FUNCTION_BLOCK NextFeedHorizon (* CAT Function Block Type *)
  (* Standard: 61499-2 *)
  (* Version 0.0, 7/15/2026, Schneider Electric, template *)
  PACKAGE SE.Nereda;
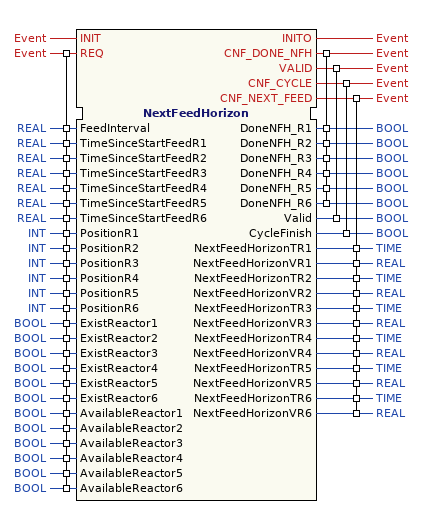
  EVENT_INPUT
    INIT;
    REQ WITH FeedInterval, TimeSinceStartFeedR1, TimeSinceStartFeedR2, TimeSinceStartFeedR3, TimeSinceStartFeedR4, TimeSinceStartFeedR5, TimeSinceStartFeedR6, PositionR1, PositionR2, PositionR3, PositionR4, PositionR5, PositionR6, ExistReactor1, ExistReactor2, ExistReactor3, ExistReactor4, ExistReactor5, ExistReactor6, AvailableReactor1, AvailableReactor2, AvailableReactor3, AvailableReactor4, AvailableReactor5, AvailableReactor6;
  END_EVENT
  EVENT_OUTPUT
    INITO;
    CNF_DONE_NFH WITH DoneNFH_R6, DoneNFH_R1, DoneNFH_R2, DoneNFH_R3, DoneNFH_R4, DoneNFH_R5;
    VALID WITH Valid; (* Execution Confirmation *)
    CNF_CYCLE WITH CycleFinish; (* Execution Confirmation *)
    CNF_NEXT_FEED WITH NextFeedHorizonTR1, NextFeedHorizonTR2, NextFeedHorizonTR3, NextFeedHorizonTR4, NextFeedHorizonTR5, NextFeedHorizonTR6, NextFeedHorizonVR1, NextFeedHorizonVR2, NextFeedHorizonVR3, NextFeedHorizonVR4, NextFeedHorizonVR5, NextFeedHorizonVR6; (* Execution Confirmation of current and total device operation duration *)
  END_EVENT
  VAR_INPUT
    FeedInterval : REAL;
    TimeSinceStartFeedR1 : REAL;
    TimeSinceStartFeedR2 : REAL;
    TimeSinceStartFeedR3 : REAL;
    TimeSinceStartFeedR4 : REAL;
    TimeSinceStartFeedR5 : REAL;
    TimeSinceStartFeedR6 : REAL;
    PositionR1 : INT;
    PositionR2 : INT;
    PositionR3 : INT;
    PositionR4 : INT;
    PositionR5 : INT;
    PositionR6 : INT;
    ExistReactor1 : BOOL;
    ExistReactor2 : BOOL;
    ExistReactor3 : BOOL;
    ExistReactor4 : BOOL;
    ExistReactor5 : BOOL;
    ExistReactor6 : BOOL;
    AvailableReactor1 : BOOL;
    AvailableReactor2 : BOOL;
    AvailableReactor3 : BOOL;
    AvailableReactor4 : BOOL;
    AvailableReactor5 : BOOL;
    AvailableReactor6 : BOOL;
  END_VAR
  VAR_OUTPUT
    DoneNFH_R1 : BOOL;
    DoneNFH_R2 : BOOL;
    DoneNFH_R3 : BOOL;
    DoneNFH_R4 : BOOL;
    DoneNFH_R5 : BOOL;
    DoneNFH_R6 : BOOL;
    Valid : BOOL;
    CycleFinish : BOOL;
    NextFeedHorizonTR1 : TIME;
    NextFeedHorizonVR1 : REAL;
    NextFeedHorizonTR2 : TIME;
    NextFeedHorizonVR2 : REAL;
    NextFeedHorizonTR3 : TIME;
    NextFeedHorizonVR3 : REAL;
    NextFeedHorizonTR4 : TIME;
    NextFeedHorizonVR4 : REAL;
    NextFeedHorizonTR5 : TIME;
    NextFeedHorizonVR5 : REAL;
    NextFeedHorizonTR6 : TIME;
    NextFeedHorizonVR6 : REAL;
  END_VAR
  (* 01 - FUNCTIONNAL INPUT INTERFACE *)
  (* 00 - INITIALIZATION *)
  (* 05 - LOGIC *)
  (* 03 - FIELD INTERFACE *)
  (* 02 - FUNCTIONNAL OUTPUT INTERFACE *)
  (* Logic *)
  (* 04 - CHILDREN *)
  (* 4A - TYPICALS *)
  (* 06 - HMI INTERFACE *)
  FBS
    NextFeedHorizon : NextFeedHorizonCalc;
    REAL_TIME : REAL2TIME_8;
    IThis : NextFeedHorizon_HMI(QI := TRUE);
    ms2min : DIVIDE(pin_02E479D09E2C7EA2 := 60000);
    CycleFinishMng : AllNextFeedDone;
    CycleFinishMngSmooth : boolValueChanged;
    FeedNextHorizonDurDone : RxDone;
    SmoothDone : BoolValueChanged_6;
    CalcDoneSmooth : boolValueChanged;
  END_FBS
  EVENT_CONNECTIONS
    NextFeedHorizon.EFD8CD031C6B32D9 TO REAL_TIME.9954577AA24F9DD6;
    REQ TO ms2min.0FDF8A587C3CA146;
    ms2min.6D05A744943B688E TO NextFeedHorizon.A58B9BBDB9ECFCA5;
    SmoothDone.350834820611931F TO CalcDoneSmooth.REQ;
    FeedNextHorizonDurDone.F66E605CFBE991BE TO SmoothDone.77F8F9CFF707DAFF;
    CycleFinishMng.C7839E6909E5584F TO CycleFinishMngSmooth.REQ;
    CycleFinishMngSmooth.CHD TO CNF_CYCLE;
    INIT TO IThis.EBDA457F8F4B39EC;
    SmoothDone.350834820611931F TO IThis.91C70CF25931E11C;
    IThis.80C77422076FA241 TO INITO;
    SmoothDone.350834820611931F TO CycleFinishMng.827D9FFB0EDC0F13;
    SmoothDone.350834820611931F TO CNF_NEXT_FEED;
    SmoothDone.93AE3729A9342678 TO CNF_DONE_NFH;
    REAL_TIME.79B40746AB555956 TO FeedNextHorizonDurDone.C7D92FA891D97969;
    CalcDoneSmooth.CHD TO VALID;
  END_CONNECTIONS
  DATA_CONNECTIONS
    NextFeedHorizon.0DCC691260B3560F TO REAL_TIME.C5068E6A004DA67A;
    NextFeedHorizon.65DD9DFF0E258395 TO REAL_TIME.090CACFE48E3AA5C;
    NextFeedHorizon.563DC3E1AC221234 TO REAL_TIME.CCAE5CE14A58FFFD;
    NextFeedHorizon.4C0C80183FC55B5A TO REAL_TIME.EC24E3C1A6E6A310;
    NextFeedHorizon.B70593E6D3D95FF1 TO REAL_TIME.A9F59D487CF4DECF;
    NextFeedHorizon.65C4708021D9B2CA TO REAL_TIME.8F105E1254810899;
    NextFeedHorizon.8A408AC9522596F0 TO REAL_TIME.158B8AA7B31D2617;
    FeedInterval TO ms2min.8EF5C40F2FEA5451;
    PositionR1 TO NextFeedHorizon.7054111BE4D91EB7;
    PositionR2 TO NextFeedHorizon.0B20A0DA317A9F10;
    PositionR3 TO NextFeedHorizon.FF3C39896E6706FC;
    PositionR4 TO NextFeedHorizon.3ED1AC1F50C1DDC5;
    PositionR5 TO NextFeedHorizon.0537CBAEFE3E33F0;
    PositionR6 TO NextFeedHorizon.F44C736C902AD671;
    ExistReactor1 TO NextFeedHorizon.9A5AAB4E801C2CA4;
    ExistReactor2 TO NextFeedHorizon.DE964A829D17457B;
    ExistReactor3 TO NextFeedHorizon.68ED98420115DCB8;
    ExistReactor4 TO NextFeedHorizon.F91E650BB68991E6;
    ExistReactor5 TO NextFeedHorizon.73BF5DEC82E9482C;
    ExistReactor6 TO NextFeedHorizon.4B5EC10E0DC11F17;
    AvailableReactor1 TO NextFeedHorizon.DDB39E45EFCED8D8;
    AvailableReactor2 TO NextFeedHorizon.534818A7890109B2;
    AvailableReactor3 TO NextFeedHorizon.BEF93F1F81559DBD;
    AvailableReactor4 TO NextFeedHorizon.F7E0AE6BB8054480;
    AvailableReactor5 TO NextFeedHorizon.EB124F6B538ADD55;
    AvailableReactor6 TO NextFeedHorizon.B60357D18066DF0E;
    FeedNextHorizonDurDone.C98FDEA92D397108 TO DoneNFH_R1;
    FeedNextHorizonDurDone.2D4EC85CE11C4908 TO DoneNFH_R2;
    FeedNextHorizonDurDone.1B935CA99D34F379 TO DoneNFH_R3;
    FeedNextHorizonDurDone.97AF662E25430824 TO DoneNFH_R4;
    FeedNextHorizonDurDone.2A3F8F868022774B TO DoneNFH_R5;
    FeedNextHorizonDurDone.BCD0027C2A299157 TO DoneNFH_R6;
    PositionR1 TO FeedNextHorizonDurDone.D7556D6059D49CA6;
    PositionR2 TO FeedNextHorizonDurDone.326938D5208F6438;
    PositionR3 TO FeedNextHorizonDurDone.3F16E00CE4743B15;
    PositionR4 TO FeedNextHorizonDurDone.EE8CD69E0821CD9B;
    PositionR5 TO FeedNextHorizonDurDone.F419CEC147F957E5;
    PositionR6 TO FeedNextHorizonDurDone.D6B3B13ABFD248A5;
    ms2min.E78A8A65D4120686 TO NextFeedHorizon.C779B02CD721992D;
    CalcDoneSmooth.Output TO Valid;
    FeedNextHorizonDurDone.C98FDEA92D397108 TO SmoothDone.25B5287A5784F3EC;
    FeedNextHorizonDurDone.2D4EC85CE11C4908 TO SmoothDone.4ABB3F1062775F74;
    FeedNextHorizonDurDone.1B935CA99D34F379 TO SmoothDone.113D29D71E6DF4C2;
    FeedNextHorizonDurDone.97AF662E25430824 TO SmoothDone.0BC4334F5BE263F8;
    FeedNextHorizonDurDone.2A3F8F868022774B TO SmoothDone.FB0E6D999B27FA12;
    FeedNextHorizonDurDone.BCD0027C2A299157 TO SmoothDone.552C61FEC6B42E99;
    CycleFinishMng.983FA8826EEC6CED TO CycleFinishMngSmooth.Input;
    CycleFinishMngSmooth.Output TO CycleFinish;
    PositionR1 TO CycleFinishMng.242371E86B1FA6FA;
    PositionR2 TO CycleFinishMng.99E9230851F158B0;
    PositionR3 TO CycleFinishMng.D2F022346EC536CC;
    PositionR4 TO CycleFinishMng.8B717B51BDCFBA56;
    PositionR5 TO CycleFinishMng.3099CDB384ACB380;
    PositionR6 TO CycleFinishMng.E2C863F1948F207D;
    TimeSinceStartFeedR1 TO NextFeedHorizon.02EE639E4A36A4E1;
    TimeSinceStartFeedR2 TO NextFeedHorizon.F586E04D8C89DEA6;
    TimeSinceStartFeedR3 TO NextFeedHorizon.AD55B2D2D554E6EC;
    TimeSinceStartFeedR4 TO NextFeedHorizon.3EBC8C13DE9A2146;
    TimeSinceStartFeedR5 TO NextFeedHorizon.C0E7B53A76514D03;
    TimeSinceStartFeedR6 TO NextFeedHorizon.DA82A5DC8F464219;
    NextFeedHorizon.65DD9DFF0E258395 TO FeedNextHorizonDurDone.860731667DF4D873;
    NextFeedHorizon.563DC3E1AC221234 TO FeedNextHorizonDurDone.14E12A3D8BF091C1;
    NextFeedHorizon.4C0C80183FC55B5A TO FeedNextHorizonDurDone.65C1CB388B57E6E2;
    NextFeedHorizon.B70593E6D3D95FF1 TO FeedNextHorizonDurDone.701DDBE1ED42FA98;
    NextFeedHorizon.65C4708021D9B2CA TO FeedNextHorizonDurDone.EF0FAC30F2F9F8D1;
    NextFeedHorizon.4F3E4C31A73CCE46 TO FeedNextHorizonDurDone.16D724347BCF5F1C;
    REAL_TIME.E4F2EB0AA0B91A9A TO NextFeedHorizonTR1;
    REAL_TIME.E201E7048FBB0948 TO NextFeedHorizonTR2;
    REAL_TIME.94DB832B06EEF2E6 TO NextFeedHorizonTR3;
    REAL_TIME.0CAC84E6FA7FE341 TO NextFeedHorizonTR4;
    REAL_TIME.422343454C5D1A84 TO NextFeedHorizonTR5;
    REAL_TIME.1ACEF24FC515D2E5 TO NextFeedHorizonTR6;
    NextFeedHorizon.65DD9DFF0E258395 TO NextFeedHorizonVR1;
    NextFeedHorizon.563DC3E1AC221234 TO NextFeedHorizonVR2;
    NextFeedHorizon.4C0C80183FC55B5A TO NextFeedHorizonVR3;
    NextFeedHorizon.B70593E6D3D95FF1 TO NextFeedHorizonVR4;
    NextFeedHorizon.65C4708021D9B2CA TO NextFeedHorizonVR5;
    NextFeedHorizon.4F3E4C31A73CCE46 TO NextFeedHorizonVR6;
    REAL_TIME.E4F2EB0AA0B91A9A TO IThis.DFC524D1F90A31A2;
    REAL_TIME.E201E7048FBB0948 TO IThis.24A26F49321919FA;
    REAL_TIME.94DB832B06EEF2E6 TO IThis.60A8AE8F5819AE1D;
    REAL_TIME.0CAC84E6FA7FE341 TO IThis.F10A3460FD914C2A;
    REAL_TIME.422343454C5D1A84 TO IThis.D6114B476C21EF4F;
    REAL_TIME.1ACEF24FC515D2E5 TO IThis.16ADDB5C293C7ACC;
    SmoothDone.AA81B8787A42C5C8 TO CycleFinishMng.A2F8E220DCBA9D90;
    SmoothDone.9956B7B3B3929CFE TO CycleFinishMng.B35D19D9BAD128AE;
    SmoothDone.0578107E6CFA5800 TO CycleFinishMng.8BC1271916155A47;
    SmoothDone.167BD6731FEB1D53 TO CycleFinishMng.559D0A9CA9501416;
    SmoothDone.1AB852B2890146E4 TO CycleFinishMng.25D8CA1F5633D382;
    SmoothDone.6C1C82B2CFBF666D TO CycleFinishMng.71B0125028A105BD;
    NextFeedHorizon.3174B0E2BA0493C7 TO CalcDoneSmooth.Input;
  END_CONNECTIONS
END_FUNCTION_BLOCK
